Yaskawa INFORM job: trapez2_21_12_2023.JBI

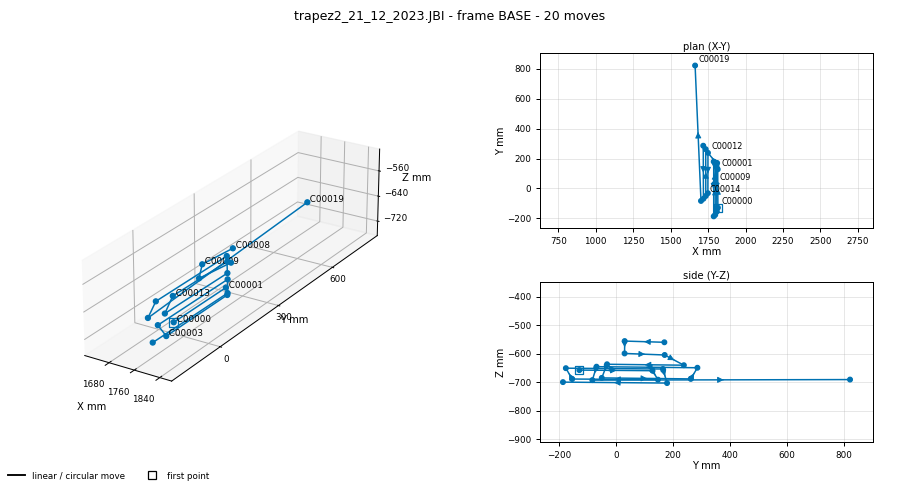
[picture p0: tool path of trapez2_21_12_2023.JBI in frame BASE, 20 of 23 moves have a stored position in this frame; points joined in program order, loops and branches not executed]
/JOB
//NAME trapez2_21_12_2023
//POS
///NPOS 20,0,20,0,0,0
///TOOL 0
///POSTYPE BASE
///RECTAN
///RCONF 0,0,0,0,0,0,0,0,0,0,0,0,0,0,0,0,0,0,0,0,0,0,0,0
C00000=1815.304188,-128.519305,-657.253016,175.000000,-77.711495,-5.000000
C00001=1814.135078,128.025728,-659.347607,175.000000,-77.711495,-5.000000
C00002=1806.410959,147.072733,-690.866273,175.000000,-77.711495,-5.000000
C00003=1808.363202,-153.857036,-688.535839,175.000000,-77.711495,-5.000000
C00004=1797.473467,-175.934668,-650.533567,175.000000,-77.711495,-5.000000
C00005=1796.616563,164.548873,-653.464796,175.000000,-77.711495,-5.000000
C00006=1787.281925,178.967541,-702.738008,175.000000,-77.711495,-5.000000
C00007=1787.349402,-186.058807,-699.410079,180.000000,-60.000000,0.000000
C00008=1810.360293,169.586584,-559.727385,-175.000000,-72.399695,-5.000000
C00009=1802.059034,30.358439,-555.463678,-175.000000,-72.399695,-5.000000
C00010=1791.841734,30.020743,-598.831541,-175.000000,-72.399695,-5.000000
C00011=1803.718751,170.637223,-604.245821,-175.000000,-72.399695,-5.000000
C00012=1748.913469,237.932804,-640.107019,-175.000000,-72.399695,-5.000000
C00013=1748.374260,-31.495782,-636.781000,-175.000000,-72.399695,-5.000000
C00014=1734.511209,-50.004412,-684.625325,-175.000000,-72.399695,-5.000000
C00015=1734.016962,262.240151,-688.124875,-175.000000,-72.399695,-5.000000
C00016=1717.502537,285.434002,-649.013909,-175.000000,-72.399695,-5.000000
C00017=1718.770980,-68.395206,-645.273002,-175.000000,-72.399695,-5.000000
C00018=1702.452961,-83.046273,-692.383722,-175.000000,-72.399695,-5.000000
C00019=1663.129147,820.734611,-690.492383,180.000000,-60.000000,0.000000
///POSTYPE PULSE
///PULSE
EC00000=5120.0
EC00001=5120.0
EC00002=5120.0
EC00003=5120.0
EC00004=5120.0
EC00005=5120.0
EC00006=5120.0
EC00007=5120.0
EC00008=188416.0
EC00009=188416.0
EC00010=188416.0
EC00011=188416.0
EC00012=188416.0
EC00013=188416.0
EC00014=188416.0
EC00015=188416.0
EC00016=188416.0
EC00017=188416.0
EC00018=188416.0
EC00019=188416.0
//INST
///DATE 2023/07/21 16:08
///ATTR SC,RW,RJ
////FRAME BASE
///GROUP1 RB1,ST1
NOP
MOVJ P009 EX000 VJ=15.00
MOVJ C00000 EC00000 VJ=15.0
CALL JOB:SPYON
MOVL C00001 EC00001 V=150.0
MOVL C00002 EC00002 V=150.0
MOVL C00003 EC00003 V=150.0
MOVL C00004 EC00004 V=150.0
MOVL C00005 EC00005 V=150.0
MOVL C00006 EC00006 V=150.0
MOVL C00007 EC00007 V=150.0
CALL JOB:SPYOF
MOVJ P009 VJ=15.00
MOVJ C00008 EC00008 VJ=15.0
CALL JOB:SPYON
MOVL C00009 EC00009 V=150.0
MOVL C00010 EC00010 V=150.0
MOVL C00011 EC00011 V=150.0
MOVL C00012 EC00012 V=150.0
MOVL C00013 EC00013 V=150.0
MOVL C00014 EC00014 V=150.0
MOVL C00015 EC00015 V=150.0
MOVL C00016 EC00016 V=150.0
MOVL C00017 EC00017 V=150.0
MOVL C00018 EC00018 V=150.0
MOVL C00019 EC00019 V=150.0
CALL JOB:SPYOF
MOVJ P009 VJ=15.00
END
